# EPICS substitutions: ek9000App/Db/EL1202.substitutions
file EL1202.template
{ 	pattern
	{
		TERMINAL,

	}
	{
	}
}
